{attribute addProperty BoxType "EK1122-0000-0018"}
{attribute addProperty Id "Beckhoff_EL15xxsub_EK1100EK1100_179A0949162"}
{attribute addProperty CRC "1353942506"}
{attribute addProperty SizeInBites "16"}
{attribute addProperty SizeInBytes "2"}
TYPE Beckhoff_EL15xxEK1122_50B385EA EXTENDS EK1122_179A0949 :
STRUCT
	{attribute addProperty Name "Beckhoff_EL15xxsub_EK1100"}
	Beckhoff_EL15xxsub_EK1100 : EK1100_179A0949;
END_STRUCT
END_TYPE

(* stored: Version 1.2.0.0, ProductVersion 3.1.4024.9
   DUT Beckhoff_EL15xxEK1122_50B385EA: Id {112681e5-91dd-4998-96cc-f3e86677dd22} *)
